{attribute 'qualified_only'}
VAR_GLOBAL
END_VAR

(* stored: Version 1.1.0.1, ProductVersion 3.1.4022.7
   GVL GVL_04_Auto_Other: Id {12eff243-9d24-4734-84dd-ba927f45894e} *)
